Staubli VAL3: Form_PattenS.pgx

public program Form_PattenS(string x_sTitle, string x_sLeftList, string x_sBottomList)
  local num l_nIndex
  local string l_sBuff[9]
  local bool l_bRes
  local string l_sBot[9]
begin
    //****************************************************************
  //***************************************************************
  //函数名称：pagePatten1s
  //用途：  用于图形显示
  //创建日期：2013.02.18
  //作者：
  //联系方式：
  //备注：
  //版本修改说明：
  //图形类型
  //                   100%
  //=========标题================
  //
  //F1->文字1
  //F2->文字2
  //F3->文字3
  //F4->文字4
  //F5->文字5
  //F6->文字6
  //F7->文字7


  //文字  文字  文字 文字 文字 文字 文字 文字
  //****************************************************************
  //*****************************************************************





  //清空
  cls()

  //标题
  title(x_sTitle)

  //把字符串给分开，使用,作为分隔符
  call Str_SplitComma(l_bRes,x_sLeftList,l_sBuff)
  if !l_bRes
    return
  endIf



  //把字符串给分开，使用,作为分隔符
  call  Str_SplitComma(l_bRes,x_sBottomList,l_sBot)
  if !l_bRes
    return
  endIf


  call Form_Patten(x_sTitle,l_sBuff,l_sBot)


end
